(* PLC project Tc2_Utilities.FB_GetVolumeId Demo, tc3-libraries-kb TwinCAT 3.1 *)
(* stored: creationDateTime 2026-05-11T00:00:00, modificationDateTime 2026-05-11T00:00:00 *)

PROGRAM P_Demo_FB_GetVolumeId
  VAR
    fbFB_GetVolumeId : FB_GetVolumeId;  (* FB_GetVolumeId 实例 *)
    bRead : BOOL := FALSE;
    volumeId : GUID;
    bBusy_ : BOOL;
    bErrFlag : BOOL;
    nErrCode : UDINT;
  END_VAR

// =============================================================================
// 场景：读卷 ID 用作 License 硬件指纹。
// 价值：比 SystemID 重装抗性更好。
// 验证：触发后 volumeId 装载非零值；与 Windows `vol C:` 命令显示一致。
// 验证步骤：
//   1. 右键 PLC 项目 → Import PLCopenXML → 选本文件
//   2. 引用 Tc2_Utilities（References → Add library）
//   3. 编译 → 登录 → 运行；按上方『验证』行的指示在线写值观察
// =============================================================================

fbFB_GetVolumeId(
    bExecute := bRead,
    tTimeout := DEFAULT_ADS_TIMEOUT,
    volumeId => volumeId,
    bBusy => bBusy_,
    bErr => bErrFlag,
    nErrId => nErrCode
);
END_PROGRAM
